(* PLC project Generated.project, CODESYS CODESYS V3.5 SP19 Patch 1 *)
(* stored: creationDateTime 2026-09-06T13:00:42.361171, modificationDateTime 2026-09-06T13:00:42.361171 *)

(* ======================================================================= ⚙️ FB_Ramp — Rampe d'accélération et décélération asymétrique ─────────────────────────────────────────────────────────────── 🎯 Rôle : Limitation de variation anti-à-coups (%/s) sur signal analogique 🔒 Polarité : Distingue l'éloignement de zéro (Accel) et le retour à zéro (Decel) 📄 Doc métier : DOC/AF/AF_Partie-11_Fonction_Translation_v2.3.md §1 (TC-P11-040) ======================================================================= *)
FUNCTION_BLOCK FB_Ramp
  VAR_INPUT
    Target : REAL;  (* === CONSIGNES ET TAUX DE RAMPE === --> [CMD] Valeur cible visee (-100.0..+100.0 %) *)
    AccelRate : REAL;  (* --> [CFG] Taux d'acceleration (%/s) *)
    DecelRate : REAL;  (* --> [CFG] Taux de deceleration (%/s) *)
    CycleTimeS : REAL;  (* --> [CFG] Temps de cycle reel en secondes (dt) *)
  END_VAR
  VAR_OUTPUT
    Current : REAL;  (* === VALEUR RAMPEE === <-- [STAT] Valeur courante amortie (-100.0..+100.0 %) *)
  END_VAR
  VAR
    StepX : REAL;  (* === CALCULS INTERNES === . [LOC] Pas de variation pour le cycle courant *)
    TargetLimited : REAL;  (* . [LOC] Cible bornee a [-100.0, +100.0] *)
  END_VAR

            

// Détection du comportement (Accélération vs Décélération)
// Classification par CÔTÉ DE ZÉRO + sens de déplacement, plus par signe brut de Target seul
// (robuste à une traversée de zéro rapide).
// 🛡️ Garde-fou : la rampe ne sort jamais de la plage normalisée ±100 %.
TargetLimited := LIMIT(-100.0, Target, 100.0);
Current := LIMIT(-100.0, Current, 100.0);

IF (Current >= 0.0 AND TargetLimited >= Current) OR (Current <= 0.0 AND TargetLimited <= Current) THEN
    StepX := AccelRate * CycleTimeS; // S'éloigne du zéro (reste du même côté, va plus loin)
ELSE
    StepX := DecelRate * CycleTimeS; // Retourne vers zéro, ou le traverse vers l'autre signe
END_IF;

// Application de la rampe
IF Current < TargetLimited THEN
    Current := Current + StepX;
    IF Current > TargetLimited THEN Current := TargetLimited; END_IF;
ELSIF Current > TargetLimited THEN
    Current := Current - StepX;
    IF Current < TargetLimited THEN Current := TargetLimited; END_IF;
END_IF;

// 🛡️ Limitation finale : même une valeur d'état déjà corrompue reste bornée.
Current := LIMIT(-100.0, Current, 100.0);

          
END_FUNCTION_BLOCK
